{attribute 'linkalways'} 
{attribute 'no_explicit_call' := 'This FB is a CLASS and must be accessed using methods or properties'}
{attribute 'enable_dynamic_creation'}
FUNCTION_BLOCK AutomaticCyclicCall EXTENDS Instance IMPLEMENTS I_CyclicInstance
VAR
	membership : GlobalInstanceMembership(THIS^);
	_cyclicInstanceCallback : CyclicCallback(0);
END_VAR

PROPERTY PUBLIC CyclicInstanceCallback : I_Callback
GET
CyclicInstanceCallback := _cyclicInstanceCallback;
END_GET
END_PROPERTY

METHOD FB_init : BOOL
VAR_INPUT
	bInitRetains : BOOL; // if TRUE, the retain variables are initialized (warm start / cold start)
	bInCopyCode : BOOL;  // if TRUE, the instance afterwards gets moved into the copy code (online change)
	Target : I_CyclicCalled;
END_VAR
_cyclicInstanceCallback.Target := Target;
membership.Join();
END_METHOD

END_FUNCTION_BLOCK

(* stored: Version 1.1.0.1, ProductVersion 3.1.4024.12
   POU AutomaticCyclicCall: Id {325a7cf6-0682-034f-22d2-c8731548a9cb}, SpecialFunc None
   Folder Constructor: Id {b2968c6c-4bed-0eeb-1245-541c508e3819}
   Property CyclicInstanceCallback: Id {a3ba8d9f-66eb-0552-1a3a-496ae1cfbc6d}
   Get Get: Id {ba8e72c7-0da0-0f61-0d7f-3a3f2aee5e0b}
   Method FB_init: Id {56b01ec9-2684-057b-065c-215e1e78c1f3} *)
